// TIA Portal V20 export
VAR_GLOBAL   // PLC tag table "BarcodeReader_DP1"
   "DP1-TriggerEnable" AT %Q81.0 : Bool;
   "DP1-Trigger" AT %Q81.1 : Bool;
   "DP1-TriggerReady" AT %I87.0 : Bool;
   "DP1-TriggerAck" AT %I87.1 : Bool;
   "DP1-Acquiring" AT %I87.2 : Bool;
   "DP1-MissedAcq" AT %I87.3 : Bool;
   "DP1-TriggerID" AT %IW88 : Word;
   "DP1-BufferResultsEnable" AT %Q82.0 : Bool;
   "DP1-ResultsAck" AT %Q82.1 : Bool;
   "DP1-Decoding" AT %I90.0 : Bool;
   "DP1-Decode Complete" AT %I90.1 : Bool;
   "DP1-Results Buffer Overrun" AT %I90.2 : Bool;
   "DP1-Results Available" AT %I90.3 : Bool;
   "DP1-General Fault" AT %I90.7 : Bool;
   "DP1-Train Code" AT %Q83.0 : Bool;
   "DP1-Train Match String" AT %Q83.1 : Bool;
   "DP1-Train Focus" AT %Q83.2 : Bool;
   "DP1-Train Brightness" AT %Q83.3 : Bool;
   "DP1-Untrain" AT %Q83.4 : Bool;
   "DP1-Execute DMCC" AT %Q83.6 : Bool;
   "DP1-Set Match String" AT %Q83.7 : Bool;
   "DP1-Train Code Ack" AT %I91.0 : Bool;
   "DP1-Train Match String Ack" AT %I91.1 : Bool;
   "DP1-Train Focus Ack" AT %I91.2 : Bool;
   "DP1-Train Brightness Ack" AT %I91.3 : Bool;
   "DP1-Untrain Ack" AT %I91.4 : Bool;
   "DP1-Execute DMCC Ack" AT %I91.6 : Bool;
   "DP1-Set Match String Ack" AT %I91.7 : Bool;
   "DP1-UserData Option" AT %QW84 : Word;
   "DP1-UserData Length" AT %QW86 : Word;
   "DP1-UserData[0]" AT %QB88 : Byte;
   "DP1-UserData[1]" AT %QB89 : Byte;
   "DP1-UserData[2]" AT %QB90 : Byte;
   "DP1-UserData[3]" AT %QB91 : Byte;
   "DP1-UserData[4]" AT %QB92 : Byte;
   "DP1-UserData[5]" AT %QB93 : Byte;
   "DP1-UserData[6]" AT %QB94 : Byte;
   "DP1-UserData[7]" AT %QB95 : Byte;
   "DP1-UserData[8]" AT %QB96 : Byte;
   "DP1-UserData[9]" AT %QB97 : Byte;
   "DP1-UserData[10]" AT %QB98 : Byte;
   "DP1-UserData[11]" AT %QB99 : Byte;
   "DP1-UserData[12]" AT %QB100 : Byte;
   "DP1-UserData[13]" AT %QB101 : Byte;
   "DP1-UserData[14]" AT %QB102 : Byte;
   "DP1-UserData[15]" AT %QB103 : Byte;
   "DP1-ResultID" AT %IW92 : Word;
   "DP1-Result Code" AT %IW95 : Word;
   "DP1-Read / No Read" AT %I95.0 : Bool;
   "DP1-Validated / Not Validated" AT %I95.1 : Bool;
   "DP1-Verified / Not Verified" AT %I95.2 : Bool;
   "DP1-Acquisition Trigger Overrun" AT %I95.3 : Bool;
   "DP1-Acquisition Buffer Overflow" AT %I95.4 : Bool;
   "DP1-Result Extended" AT %IW96 : Word;
   "DP1-Result Length" AT %IW98 : Word;
   "DP1-InspectionResults[0]" AT %IB100 : Byte;
   "DP1-InspectionResults[1]" AT %IB101 : Byte;
   "DP1-InspectionResults[2]" AT %IB102 : Byte;
   "DP1-InspectionResults[3]" AT %IB103 : Byte;
   "DP1-InspectionResults[4]" AT %IB104 : Byte;
   "DP1-InspectionResults[5]" AT %IB105 : Byte;
   "DP1-InspectionResults[6]" AT %IB106 : Byte;
   "DP1-InspectionResults[7]" AT %IB107 : Byte;
   "DP1-InspectionResults[8]" AT %IB108 : Byte;
   "DP1-InspectionResults[9]" AT %IB109 : Byte;
   "DP1-InspectionResults[10]" AT %IB110 : Byte;
   "DP1-InspectionResults[11]" AT %IB111 : Byte;
   "DP1-InspectionResults[12]" AT %IB112 : Byte;
   "DP1-InspectionResults[13]" AT %IB113 : Byte;
   "DP1-InspectionResults[14]" AT %IB114 : Byte;
   "DP1-InspectionResults[15]" AT %IB115 : Byte;
   "Result data_DP1" AT %I100.0 : "Global.BarCode";
   UserData_DP1 AT %Q88.0 : "Global.BarCode";
   ContinousGetResults_DP1 AT %M110.1 : Bool;
   TrainFocus_DP1 AT %M110.2 : Bool;
END_VAR
